# B&R Automation Studio project testovaci_pneu_stan
Automation Studio 4.9

## Configuration Config1

### Acp10map.ncm - 4PPC70_0702_20B/Motion/Acp10map.ncm
```
NcMapping (NcSwId=Acp10)
  NcObject gAxis01 (ModuleId=8V1010.50-2, Type=ncAXIS, Channel=1, AcoposSimulation=Off, InitParameter=gAxis01i, AcoposParameter=gAxis01a, Disabled=FALSE, ModuleDisabled=FALSE)
  NcObject 8V1010.50-2_ncV_AXIS1 (ModuleId=8V1010.50-2, Type=ncV_AXIS, Channel=1, Disabled=TRUE, ModuleDisabled=FALSE)
  NcObject gAxis02 (ModuleId=8V1010.50-2a, Type=ncAXIS, Channel=1, AcoposSimulation=Off, InitParameter=gAxis02i, AcoposParameter=gAxis02a, Disabled=FALSE, ModuleDisabled=FALSE)
  NcObject 8V1010.50-2a_ncV_AXIS1 (ModuleId=8V1010.50-2a, Type=ncV_AXIS, Channel=1, Disabled=TRUE, ModuleDisabled=FALSE)
```

## Logical view

### Library Logical/Libraries/pomoc_lib

#### pomoc_lib.fun
```iecst
FUNCTION_BLOCK cyklovac_b
	VAR_INPUT
		ssMethodType :  SINT;
		krok_tlaku :  REAL :=  0; (*riadok matice zasobujucej cyklovac*)
	END_VAR
	VAR_OUTPUT
		tlak_blue_1 :  REAL :=  0; (*blue_tlak*)
		tlak_green_1 :  REAL :=  0; (**)
		tlak_yellow_1 :  REAL :=  0; (**)
	END_VAR
	VAR
		bur_B_cyklovac_BB_T :  B_cyklovac_BB_T;
		bur_cyklovac_BB :  tag_RTM_cyklovac_BB_T;
	END_VAR
END_FUNCTION_BLOCK
```

#### cyklovac_BB.h
```c
/*
 * cyklovac_BB.h
 *
 * Academic License - for use in teaching, academic research, and meeting
 * course requirements at degree granting institutions only.  Not for
 * government, commercial, or other organizational use.
 *
 * Code generation for model "cyklovac_BB".
 *
 * Model version              : 1.8
 * Simulink Coder version : 9.6 (R2021b) 14-May-2021
 * C source code generated on : Thu Mar 17 07:18:42 2022
 *
 * Target selection: bur_grt.tlc
 * Note: GRT includes extra infrastructure and instrumentation for prototyping
 * Embedded hardware selection: Intel->x86/Pentium
 * Code generation objectives: Unspecified
 * Validation result: Not run
 */

#ifndef RTW_HEADER_cyklovac_BB_h_
#define RTW_HEADER_cyklovac_BB_h_
#include <stddef.h>
#include <string.h>
#ifndef cyklovac_BB_COMMON_INCLUDES_
#define cyklovac_BB_COMMON_INCLUDES_
#include <stdlib.h>
#include "rtwtypes.h"
#include "rtw_continuous.h"
#include "rtw_solver.h"
#endif                                 /* cyklovac_BB_COMMON_INCLUDES_ */

#include "cyklovac_BB_types.h"
#include "pomoc_lib.h"
/* Beginning of Dynamic TypeDefs: */
/* End of Dynamic TypeDefs: */
#ifndef MIN
#define MIN(a,b)	((a) < (b) ? (a) : (b))
#endif

#ifndef MAX
#define MAX(a,b)	((a) > (b) ? (a) : (b))
#endif

#ifndef AST_ROUND
#define AST_ROUND(x) ((x)>=0?(long long)((x)+0.5):(long long)((x)-0.5))
#endif

/* Shared type includes */
#include "multiword_types.h"
#include "rt_defines.h"

/* Macros for accessing real-time model data structure */
#ifndef rtmGetBlockIO
#define rtmGetBlockIO(rtm)             ((rtm)->blockIO)
#endif

#ifndef rtmSetBlockIO
#define rtmSetBlockIO(rtm, val)        ((rtm)->blockIO = (val))
#endif

#ifndef rtmGetErrorStatus
#define rtmGetErrorStatus(rtm)         ((rtm)->errorStatus)
#endif

#ifndef rtmSetErrorStatus
#define rtmSetErrorStatus(rtm, val)    ((rtm)->errorStatus = (val))
#endif

#define cyklovac_BB_M_TYPE             RT_MODEL_cyklovac_BB_T

/* Block signals (default storage) */

/* Constant parameters (default storage) */

/* Real-time Model Data Structure */

/* External data declarations for dependent source files */
extern const char *RT_MEMORY_ALLOCATION_ERROR;

/* Constant parameters (default storage) */
extern const ConstP_cyklovac_BB_T cyklovac_BB_ConstP;

/* Model entry point functions */
extern void cyklovac_BB_initializeMemory(RT_MODEL_cyklovac_BB_T * const cyklovac_BB_M, struct cyklovac_b* inst);
extern void cyklovac_BB_initialize(RT_MODEL_cyklovac_BB_T *const cyklovac_BB_M, struct cyklovac_b* inst);
extern void cyklovac_BB_step(RT_MODEL_cyklovac_BB_T *const cyklovac_BB_M, struct cyklovac_b* inst);
extern void cyklovac_BB_terminate(RT_MODEL_cyklovac_BB_T * cyklovac_BB_M, struct cyklovac_b* inst);

/*-
 * The generated code includes comments that allow you to trace directly
 * back to the appropriate location in the model.  The basic format
 * is <system>/block_name, where system is the system number (uniquely
 * assigned by Simulink) and block_name is the name of the block.
 *
 * Use the MATLAB hilite_system command to trace the generated code back
 * to the model.  For example,
 *
 * hilite_system('<S3>')    - opens system 3
 * hilite_system('<S3>/Kp') - opens and selects block Kp which resides in S3
 *
 * Here is the system hierarchy for this model
 *
 * '<Root>' : 'cyklovac_BB'
 * '<S1>'   : 'cyklovac_BB/MATLAB Function'
 */
#endif                                 /* RTW_HEADER_cyklovac_BB_h_ */
```

#### cyklovac_BB_types.h
```c
/*
 * cyklovac_BB_types.h
 *
 * Academic License - for use in teaching, academic research, and meeting
 * course requirements at degree granting institutions only.  Not for
 * government, commercial, or other organizational use.
 *
 * Code generation for model "cyklovac_BB".
 *
 * Model version              : 1.8
 * Simulink Coder version : 9.6 (R2021b) 14-May-2021
 * C source code generated on : Thu Mar 17 07:18:42 2022
 *
 * Target selection: bur_grt.tlc
 * Note: GRT includes extra infrastructure and instrumentation for prototyping
 * Embedded hardware selection: Intel->x86/Pentium
 * Code generation objectives: Unspecified
 * Validation result: Not run
 */

#ifndef RTW_HEADER_cyklovac_BB_types_h_
#define RTW_HEADER_cyklovac_BB_types_h_

/* Model Code Variants */

/* Forward declaration for rtModel */

#endif                                 /* RTW_HEADER_cyklovac_BB_types_h_ */
```

#### multiword_types.h
```c
/*
 * multiword_types.h
 *
 * Academic License - for use in teaching, academic research, and meeting
 * course requirements at degree granting institutions only.  Not for
 * government, commercial, or other organizational use.
 *
 * Code generation for model "cyklovac_BB".
 *
 * Model version              : 1.8
 * Simulink Coder version : 9.6 (R2021b) 14-May-2021
 * C source code generated on : Thu Mar 17 07:18:42 2022
 *
 * Target selection: bur_grt.tlc
 * Note: GRT includes extra infrastructure and instrumentation for prototyping
 * Embedded hardware selection: Intel->x86/Pentium
 * Code generation objectives: Unspecified
 * Validation result: Not run
 */

#ifndef MULTIWORD_TYPES_H
#define MULTIWORD_TYPES_H
#include "rtwtypes.h"

/*
 * MultiWord supporting definitions
 */
typedef long int long_T;

/*
 * MultiWord types
 */
typedef struct {
  uint32_T chunks[2];
} int64m_T;

typedef struct {
  int64m_T re;
  int64m_T im;
} cint64m_T;

typedef struct {
  uint32_T chunks[2];
} uint64m_T;

typedef struct {
  uint64m_T re;
  uint64m_T im;
} cuint64m_T;

typedef struct {
  uint32_T chunks[3];
} int96m_T;

typedef struct {
  int96m_T re;
  int96m_T im;
} cint96m_T;

typedef struct {
  uint32_T chunks[3];
} uint96m_T;

typedef struct {
  uint96m_T re;
  uint96m_T im;
} cuint96m_T;

typedef struct {
  uint32_T chunks[4];
} int128m_T;

typedef struct {
  int128m_T re;
  int128m_T im;
} cint128m_T;

typedef struct {
  uint32_T chunks[4];
} uint128m_T;

typedef struct {
  uint128m_T re;
  uint128m_T im;
} cuint128m_T;

typedef struct {
  uint32_T chunks[5];
} int160m_T;

typedef struct {
  int160m_T re;
  int160m_T im;
} cint160m_T;

typedef struct {
  uint32_T chunks[5];
} uint160m_T;

typedef struct {
  uint160m_T re;
  uint160m_T im;
} cuint160m_T;

typedef struct {
  uint32_T chunks[6];
} int192m_T;

typedef struct {
  int192m_T re;
  int192m_T im;
} cint192m_T;

typedef struct {
  uint32_T chunks[6];
} uint192m_T;

typedef struct {
  uint192m_T re;
  uint192m_T im;
} cuint192m_T;

typedef struct {
  uint32_T chunks[7];
} int224m_T;

typedef struct {
  int224m_T re;
  int224m_T im;
} cint224m_T;

typedef struct {
  uint32_T chunks[7];
} uint224m_T;

typedef struct {
  uint224m_T re;
  uint224m_T im;
} cuint224m_T;

typedef struct {
  uint32_T chunks[8];
} int256m_T;

typedef struct {
  int256m_T re;
  int256m_T im;
} cint256m_T;

typedef struct {
  uint32_T chunks[8];
} uint256m_T;

typedef struct {
  uint256m_T re;
  uint256m_T im;
} cuint256m_T;

typedef struct {
  uint32_T chunks[9];
} int288m_T;

typedef struct {
  int288m_T re;
  int288m_T im;
} cint288m_T;

typedef struct {
  uint32_T chunks[9];
} uint288m_T;

typedef struct {
  uint288m_T re;
  uint288m_T im;
} cuint288m_T;

typedef struct {
  uint32_T chunks[10];
} int320m_T;

typedef struct {
  int320m_T re;
  int320m_T im;
} cint320m_T;

typedef struct {
  uint32_T chunks[10];
} uint320m_T;

typedef struct {
  uint320m_T re;
  uint320m_T im;
} cuint320m_T;

typedef struct {
  uint32_T chunks[11];
} int352m_T;

typedef struct {
  int352m_T re;
  int352m_T im;
} cint352m_T;

typedef struct {
  uint32_T chunks[11];
} uint352m_T;

typedef struct {
  uint352m_T re;
  uint352m_T im;
} cuint352m_T;

typedef struct {
  uint32_T chunks[12];
} int384m_T;

typedef struct {
  int384m_T re;
  int384m_T im;
} cint384m_T;

typedef struct {
  uint32_T chunks[12];
} uint384m_T;

typedef struct {
  uint384m_T re;
  uint384m_T im;
} cuint384m_T;

typedef struct {
  uint32_T chunks[13];
} int416m_T;

typedef struct {
  int416m_T re;
  int416m_T im;
} cint416m_T;

typedef struct {
  uint32_T chunks[13];
} uint416m_T;

typedef struct {
  uint416m_T re;
  uint416m_T im;
} cuint416m_T;

typedef struct {
  uint32_T chunks[14];
} int448m_T;

typedef struct {
  int448m_T re;
  int448m_T im;
} cint448m_T;

typedef struct {
  uint32_T chunks[14];
} uint448m_T;

typedef struct {
  uint448m_T re;
  uint448m_T im;
} cuint448m_T;

typedef struct {
  uint32_T chunks[15];
} int480m_T;

typedef struct {
  int480m_T re;
  int480m_T im;
} cint480m_T;

typedef struct {
  uint32_T chunks[15];
} uint480m_T;

typedef struct {
  uint480m_T re;
  uint480m_T im;
} cuint480m_T;

typedef struct {
  uint32_T chunks[16];
} int512m_T;

typedef struct {
  int512m_T re;
  int512m_T im;
} cint512m_T;

typedef struct {
  uint32_T chunks[16];
} uint512m_T;

typedef struct {
  uint512m_T re;
  uint512m_T im;
} cuint512m_T;

typedef struct {
  uint32_T chunks[17];
} int544m_T;

typedef struct {
  int544m_T re;
  int544m_T im;
} cint544m_T;

typedef struct {
  uint32_T chunks[17];
} uint544m_T;

typedef struct {
  uint544m_T re;
  uint544m_T im;
} cuint544m_T;

typedef struct {
  uint32_T chunks[18];
} int576m_T;

typedef struct {
  int576m_T re;
  int576m_T im;
} cint576m_T;

typedef struct {
  uint32_T chunks[18];
} uint576m_T;

typedef struct {
  uint576m_T re;
  uint576m_T im;
} cuint576m_T;

typedef struct {
  uint32_T chunks[19];
} int608m_T;

typedef struct {
  int608m_T re;
  int608m_T im;
} cint608m_T;

typedef struct {
  uint32_T chunks[19];
} uint608m_T;

typedef struct {
  uint608m_T re;
  uint608m_T im;
} cuint608m_T;

typedef struct {
  uint32_T chunks[20];
} int640m_T;

typedef struct {
  int640m_T re;
  int640m_T im;
} cint640m_T;

typedef struct {
  uint32_T chunks[20];
} uint640m_T;

typedef struct {
  uint640m_T re;
  uint640m_T im;
} cuint640m_T;

typedef struct {
  uint32_T chunks[21];
} int672m_T;

typedef struct {
  int672m_T re;
  int672m_T im;
} cint672m_T;

typedef struct {
  uint32_T chunks[21];
} uint672m_T;

typedef struct {
  uint672m_T re;
  uint672m_T im;
} cuint672m_T;

typedef struct {
  uint32_T chunks[22];
} int704m_T;

typedef struct {
  int704m_T re;
  int704m_T im;
} cint704m_T;

typedef struct {
  uint32_T chunks[22];
} uint704m_T;

typedef struct {
  uint704m_T re;
  uint704m_T im;
} cuint704m_T;

typedef struct {
  uint32_T chunks[23];
} int736m_T;

typedef struct {
  int736m_T re;
  int736m_T im;
} cint736m_T;

typedef struct {
  uint32_T chunks[23];
} uint736m_T;

typedef struct {
  uint736m_T re;
  uint736m_T im;
} cuint736m_T;

typedef struct {
  uint32_T chunks[24];
} int768m_T;

typedef struct {
  int768m_T re;
  int768m_T im;
} cint768m_T;

typedef struct {
  uint32_T chunks[24];
} uint768m_T;

typedef struct {
  uint768m_T re;
  uint768m_T im;
} cuint768m_T;

typedef struct {
  uint32_T chunks[25];
} int800m_T;

typedef struct {
  int800m_T re;
  int800m_T im;
} cint800m_T;

typedef struct {
  uint32_T chunks[25];
} uint800m_T;

typedef struct {
  uint800m_T re;
  uint800m_T im;
} cuint800m_T;

typedef struct {
  uint32_T chunks[26];
} int832m_T;

typedef struct {
  int832m_T re;
  int832m_T im;
} cint832m_T;

typedef struct {
  uint32_T chunks[26];
} uint832m_T;

typedef struct {
  uint832m_T re;
  uint832m_T im;
} cuint832m_T;

typedef struct {
  uint32_T chunks[27];
} int864m_T;

typedef struct {
  int864m_T re;
  int864m_T im;
} cint864m_T;

typedef struct {
  uint32_T chunks[27];
} uint864m_T;

typedef struct {
  uint864m_T re;
  uint864m_T im;
} cuint864m_T;

typedef struct {
  uint32_T chunks[28];
} int896m_T;

typedef struct {
  int896m_T re;
  int896m_T im;
} cint896m_T;

typedef struct {
  uint32_T chunks[28];
} uint896m_T;

typedef struct {
  uint896m_T re;
  uint896m_T im;
} cuint896m_T;

typedef struct {
  uint32_T chunks[29];
} int928m_T;

typedef struct {
  int928m_T re;
  int928m_T im;
} cint928m_T;

typedef struct {
  uint32_T chunks[29];
} uint928m_T;

typedef struct {
  uint928m_T re;
  uint928m_T im;
} cuint928m_T;

typedef struct {
  uint32_T chunks[30];
} int960m_T;

typedef struct {
  int960m_T re;
  int960m_T im;
} cint960m_T;

typedef struct {
  uint32_T chunks[30];
} uint960m_T;

typedef struct {
  uint960m_T re;
  uint960m_T im;
} cuint960m_T;

typedef struct {
  uint32_T chunks[31];
} int992m_T;

typedef struct {
  int992m_T re;
  int992m_T im;
} cint992m_T;

typedef struct {
  uint32_T chunks[31];
} uint992m_T;

typedef struct {
  uint992m_T re;
  uint992m_T im;
} cuint992m_T;

typedef struct {
  uint32_T chunks[32];
} int1024m_T;

typedef struct {
  int1024m_T re;
  int1024m_T im;
} cint1024m_T;

typedef struct {
  uint32_T chunks[32];
} uint1024m_T;

typedef struct {
  uint1024m_T re;
  uint1024m_T im;
} cuint1024m_T;

typedef struct {
  uint32_T chunks[33];
} int1056m_T;

typedef struct {
  int1056m_T re;
  int1056m_T im;
} cint1056m_T;

typedef struct {
  uint32_T chunks[33];
} uint1056m_T;

typedef struct {
  uint1056m_T re;
  uint1056m_T im;
} cuint1056m_T;

typedef struct {
  uint32_T chunks[34];
} int1088m_T;

typedef struct {
  int1088m_T re;
  int1088m_T im;
} cint1088m_T;

typedef struct {
  uint32_T chunks[34];
} uint1088m_T;

typedef struct {
  uint1088m_T re;
  uint1088m_T im;
} cuint1088m_T;

typedef struct {
  uint32_T chunks[35];
} int1120m_T;

typedef struct {
  int1120m_T re;
  int1120m_T im;
} cint1120m_T;

typedef struct {
  uint32_T chunks[35];
} uint1120m_T;

typedef struct {
  uint1120m_T re;
  uint1120m_T im;
} cuint1120m_T;

typedef struct {
  uint32_T chunks[36];
} int1152m_T;

typedef struct {
  int1152m_T re;
  int1152m_T im;
} cint1152m_T;

typedef struct {
  uint32_T chunks[36];
} uint1152m_T;

typedef struct {
  uint1152m_T re;
  uint1152m_T im;
} cuint1152m_T;

typedef struct {
  uint32_T chunks[37];
} int1184m_T;

typedef struct {
  int1184m_T re;
  int1184m_T im;
} cint1184m_T;

typedef struct {
  uint32_T chunks[37];
} uint1184m_T;

typedef struct {
  uint1184m_T re;
  uint1184m_T im;
} cuint1184m_T;

typedef struct {
  uint32_T chunks[38];
} int1216m_T;

typedef struct {
  int1216m_T re;
  int1216m_T im;
} cint1216m_T;

typedef struct {
  uint32_T chunks[38];
} uint1216m_T;

typedef struct {
  uint1216m_T re;
  uint1216m_T im;
} cuint1216m_T;

typedef struct {
  uint32_T chunks[39];
} int1248m_T;

typedef struct {
  int1248m_T re;
  int1248m_T im;
} cint1248m_T;

typedef struct {
  uint32_T chunks[39];
} uint1248m_T;

typedef struct {
  uint1248m_T re;
  uint1248m_T im;
} cuint1248m_T;

typedef struct {
  uint32_T chunks[40];
} int1280m_T;

typedef struct {
  int1280m_T re;
  int1280m_T im;
} cint1280m_T;

typedef struct {
  uint32_T chunks[40];
} uint1280m_T;

typedef struct {
  uint1280m_T re;
  uint1280m_T im;
} cuint1280m_T;

typedef struct {
  uint32_T chunks[41];
} int1312m_T;

typedef struct {
  int1312m_T re;
  int1312m_T im;
} cint1312m_T;

typedef struct {
  uint32_T chunks[41];
} uint1312m_T;

typedef struct {
  uint1312m_T re;
  uint1312m_T im;
} cuint1312m_T;

typedef struct {
  uint32_T chunks[42];
} int1344m_T;

typedef struct {
  int1344m_T re;
  int1344m_T im;
} cint1344m_T;

typedef struct {
  uint32_T chunks[42];
} uint1344m_T;

typedef struct {
  uint1344m_T re;
  uint1344m_T im;
} cuint1344m_T;

typedef struct {
  uint32_T chunks[43];
} int1376m_T;

typedef struct {
  int1376m_T re;
  int1376m_T im;
} cint1376m_T;

typedef struct {
  uint32_T chunks[43];
} uint1376m_T;

typedef struct {
  uint1376m_T re;
  uint1376m_T im;
} cuint1376m_T;

typedef struct {
  uint32_T chunks[44];
} int1408m_T;

typedef struct {
  int1408m_T re;
  int1408m_T im;
} cint1408m_T;

typedef struct {
  uint32_T chunks[44];
} uint1408m_T;

typedef struct {
  uint1408m_T re;
  uint1408m_T im;
} cuint1408m_T;

typedef struct {
  uint32_T chunks[45];
} int1440m_T;

typedef struct {
  int1440m_T re;
  int1440m_T im;
} cint1440m_T;

typedef struct {
  uint32_T chunks[45];
} uint1440m_T;

typedef struct {
  uint1440m_T re;
  uint1440m_T im;
} cuint1440m_T;

typedef struct {
  uint32_T chunks[46];
} int1472m_T;

typedef struct {
  int1472m_T re;
  int1472m_T im;
} cint1472m_T;

typedef struct {
  uint32_T chunks[46];
} uint1472m_T;

typedef struct {
  uint1472m_T re;
  uint1472m_T im;
} cuint1472m_T;

typedef struct {
  uint32_T chunks[47];
} int1504m_T;

typedef struct {
  int1504m_T re;
  int1504m_T im;
} cint1504m_T;

typedef struct {
  uint32_T chunks[47];
} uint1504m_T;

typedef struct {
  uint1504m_T re;
  uint1504m_T im;
} cuint1504m_T;

typedef struct {
  uint32_T chunks[48];
} int1536m_T;

typedef struct {
  int1536m_T re;
  int1536m_T im;
} cint1536m_T;

typedef struct {
  uint32_T chunks[48];
} uint1536m_T;

typedef struct {
  uint1536m_T re;
  uint1536m_T im;
} cuint1536m_T;

typedef struct {
  uint32_T chunks[49];
} int1568m_T;

typedef struct {
  int1568m_T re;
  int1568m_T im;
} cint1568m_T;

typedef struct {
  uint32_T chunks[49];
} uint1568m_T;

typedef struct {
  uint1568m_T re;
  uint1568m_T im;
} cuint1568m_T;

typedef struct {
  uint32_T chunks[50];
} int1600m_T;

typedef struct {
  int1600m_T re;
  int1600m_T im;
} cint1600m_T;

typedef struct {
  uint32_T chunks[50];
} uint1600m_T;

typedef struct {
  uint1600m_T re;
  uint1600m_T im;
} cuint1600m_T;

typedef struct {
  uint32_T chunks[51];
} int1632m_T;

typedef struct {
  int1632m_T re;
  int1632m_T im;
} cint1632m_T;

typedef struct {
  uint32_T chunks[51];
} uint1632m_T;

typedef struct {
  uint1632m_T re;
  uint1632m_T im;
} cuint1632m_T;

typedef struct {
  uint32_T chunks[52];
} int1664m_T;

typedef struct {
  int1664m_T re;
  int1664m_T im;
} cint1664m_T;

typedef struct {
  uint32_T chunks[52];
} uint1664m_T;

typedef struct {
  uint1664m_T re;
  uint1664m_T im;
} cuint1664m_T;

typedef struct {
  uint32_T chunks[53];
} int1696m_T;

typedef struct {
  int1696m_T re;
  int1696m_T im;
} cint1696m_T;

typedef struct {
  uint32_T chunks[53];
} uint1696m_T;

typedef struct {
  uint1696m_T re;
  uint1696m_T im;
} cuint1696m_T;

typedef struct {
  uint32_T chunks[54];
} int1728m_T;

typedef struct {
  int1728m_T re;
  int1728m_T im;
} cint1728m_T;

typedef struct {
  uint32_T chunks[54];
} uint1728m_T;

typedef struct {
  uint1728m_T re;
  uint1728m_T im;
} cuint1728m_T;

typedef struct {
  uint32_T chunks[55];
} int1760m_T;

typedef struct {
  int1760m_T re;
  int1760m_T im;
} cint1760m_T;

typedef struct {
  uint32_T chunks[55];
} uint1760m_T;

typedef struct {
  uint1760m_T re;
  uint1760m_T im;
} cuint1760m_T;

typedef struct {
  uint32_T chunks[56];
} int1792m_T;

typedef struct {
  int1792m_T re;
  int1792m_T im;
} cint1792m_T;

typedef struct {
  uint32_T chunks[56];
} uint1792m_T;

typedef struct {
  uint1792m_T re;
  uint1792m_T im;
} cuint1792m_T;

typedef struct {
  uint32_T chunks[57];
} int1824m_T;

typedef struct {
  int1824m_T re;
  int1824m_T im;
} cint1824m_T;

typedef struct {
  uint32_T chunks[57];
} uint1824m_T;

typedef struct {
  uint1824m_T re;
  uint1824m_T im;
} cuint1824m_T;

typedef struct {
  uint32_T chunks[58];
} int1856m_T;

typedef struct {
  int1856m_T re;
  int1856m_T im;
} cint1856m_T;

typedef struct {
  uint32_T chunks[58];
} uint1856m_T;

typedef struct {
  uint1856m_T re;
  uint1856m_T im;
} cuint1856m_T;

typedef struct {
  uint32_T chunks[59];
} int1888m_T;

typedef struct {
  int1888m_T re;
  int1888m_T im;
} cint1888m_T;

typedef struct {
  uint32_T chunks[59];
} uint1888m_T;

typedef struct {
  uint1888m_T re;
  uint1888m_T im;
} cuint1888m_T;

typedef struct {
  uint32_T chunks[60];
} int1920m_T;

typedef struct {
  int1920m_T re;
  int1920m_T im;
} cint1920m_T;

typedef struct {
  uint32_T chunks[60];
} uint1920m_T;

typedef struct {
  uint1920m_T re;
  uint1920m_T im;
} cuint1920m_T;

typedef struct {
  uint32_T chunks[61];
} int1952m_T;

typedef struct {
  int1952m_T re;
  int1952m_T im;
} cint1952m_T;

typedef struct {
  uint32_T chunks[61];
} uint1952m_T;

typedef struct {
  uint1952m_T re;
  uint1952m_T im;
} cuint1952m_T;

typedef struct {
  uint32_T chunks[62];
} int1984m_T;

typedef struct {
  int1984m_T re;
  int1984m_T im;
} cint1984m_T;

typedef struct {
  uint32_T chunks[62];
} uint1984m_T;

typedef struct {
  uint1984m_T re;
  uint1984m_T im;
} cuint1984m_T;

typedef struct {
  uint32_T chunks[63];
} int2016m_T;

typedef struct {
  int2016m_T re;
  int2016m_T im;
} cint2016m_T;

typedef struct {
  uint32_T chunks[63];
} uint2016m_T;

typedef struct {
  uint2016m_T re;
  uint2016m_T im;
} cuint2016m_T;

typedef struct {
  uint32_T chunks[64];
} int2048m_T;

typedef struct {
  int2048m_T re;
  int2048m_T im;
} cint2048m_T;

typedef struct {
  uint32_T chunks[64];
} uint2048m_T;

typedef struct {
  uint2048m_T re;
  uint2048m_T im;
} cuint2048m_T;

#endif                                 /* MULTIWORD_TYPES_H */
```

#### cyklovac_BB.c
```c
/*
 * cyklovac_BB.c
 *
 * Academic License - for use in teaching, academic research, and meeting
 * course requirements at degree granting institutions only.  Not for
 * government, commercial, or other organizational use.
 *
 * Code generation for model "cyklovac_BB".
 *
 * Model version              : 1.8
 * Simulink Coder version : 9.6 (R2021b) 14-May-2021
 * C source code generated on : Thu Mar 17 07:18:42 2022
 *
 * Target selection: bur_grt.tlc
 * Note: GRT includes extra infrastructure and instrumentation for prototyping
 * Embedded hardware selection: Intel->x86/Pentium
 * Code generation objectives: Unspecified
 * Validation result: Not run
 */

#include "cyklovac_BB.h"
#include "cyklovac_BB_private.h"

/* Model step function */
void cyklovac_BB_step(RT_MODEL_cyklovac_BB_T *const cyklovac_BB_M, struct cyklovac_b* inst)
{
  B_cyklovac_BB_T *cyklovac_BB_B = cyklovac_BB_M->blockIO;

  /* S-Function (bur_in): '<Root>/Input' */
  cyklovac_BB_B->Input = inst->krok_tlaku;

  /* Gain: '<Root>/Gain' incorporates:
   *  Constant: '<Root>/Constant'
   *  MATLAB Function: '<Root>/MATLAB Function'
   */
  cyklovac_BB_B->Gain = (real32_T)cyklovac_BB_ConstP.Constant_Value[(int32_T)
    cyklovac_BB_B->Input - 1];

  /* S-Function (bur_out): '<Root>/Output' */
  inst->tlak_blue_1 = cyklovac_BB_B->Gain;

  /* Gain: '<Root>/Gain1' incorporates:
   *  Constant: '<Root>/Constant'
   *  MATLAB Function: '<Root>/MATLAB Function'
   */
  cyklovac_BB_B->Gain1 = (real32_T)cyklovac_BB_ConstP.Constant_Value[(int32_T)
    cyklovac_BB_B->Input + 783];

  /* S-Function (bur_out): '<Root>/Output1' */
  inst->tlak_green_1 = cyklovac_BB_B->Gain1;

  /* Gain: '<Root>/Gain2' incorporates:
   *  Constant: '<Root>/Constant'
   *  MATLAB Function: '<Root>/MATLAB Function'
   */
  cyklovac_BB_B->Gain2 = (real32_T)cyklovac_BB_ConstP.Constant_Value[(int32_T)
    cyklovac_BB_B->Input + 1567];

  /* S-Function (bur_out): '<Root>/Output2' */
  inst->tlak_yellow_1 = cyklovac_BB_B->Gain2;
}

/* Model initialize function */
void cyklovac_BB_initialize(RT_MODEL_cyklovac_BB_T *const cyklovac_BB_M, struct cyklovac_b* inst)
{
  UNUSED_PARAMETER(cyklovac_BB_M);
}

/* Model terminate function */
void cyklovac_BB_terminate(RT_MODEL_cyklovac_BB_T * cyklovac_BB_M, struct cyklovac_b* inst)
{}

/* Model data allocation function */
void cyklovac_BB_initializeMemory(RT_MODEL_cyklovac_BB_T* const cyklovac_BB_M, struct cyklovac_b * inst)
{
  /* block I/O */
  {
  }

  {
    B_cyklovac_BB_T *cyklovac_BB_B = cyklovac_BB_M->blockIO;

    /* block I/O */
    {
      cyklovac_BB_B->Input = 0.0F;
      cyklovac_BB_B->Gain = 0.0F;
      cyklovac_BB_B->Gain1 = 0.0F;
      cyklovac_BB_B->Gain2 = 0.0F;
    }
  }

}
```

#### cyklovac_BB_data.c
```c
/*
 * cyklovac_BB_data.c
 *
 * Academic License - for use in teaching, academic research, and meeting
 * course requirements at degree granting institutions only.  Not for
 * government, commercial, or other organizational use.
 *
 * Code generation for model "cyklovac_BB".
 *
 * Model version              : 1.8
 * Simulink Coder version : 9.6 (R2021b) 14-May-2021
 * C source code generated on : Thu Mar 17 07:18:42 2022
 *
 * Target selection: bur_grt.tlc
 * Note: GRT includes extra infrastructure and instrumentation for prototyping
 * Embedded hardware selection: Intel->x86/Pentium
 * Code generation objectives: Unspecified
 * Validation result: Not run
 */

#include "cyklovac_BB.h"
#include "cyklovac_BB_private.h"

/* Constant parameters (default storage) */
const ConstP_cyklovac_BB_T cyklovac_BB_ConstP = {
  /* Expression: tlaky_upravene
   * Referenced by: '<Root>/Constant'
   */
  { 0.25, 0.25, 0.25, 0.25, 0.25, 0.25, 0.25, 0.25, 0.25, 0.25, 0.25, 0.25, 0.25,
    0.25, 0.25, 0.25, 0.25, 0.25, 0.25, 0.25, 0.25, 0.25, 0.25, 0.25, 0.25, 0.25,
    0.25, 0.25, 0.25, 0.25, 0.25, 0.25, 0.25, 0.25, 0.25, 0.25, 0.25, 0.25, 0.25,
    0.25, 0.25, 0.25, 0.25, 0.25, 0.25, 0.25, 0.25, 0.25, 0.25, 0.25, 0.25, 0.25,
    0.25, 0.25, 0.25, 0.25, 0.25, 0.25, 0.25, 0.25, 0.25, 0.25, 0.25, 0.25, 0.25,
    0.25, 0.25, 0.25, 0.25, 0.25, 0.25, 0.25, 0.25, 0.25, 0.25, 0.25, 0.25, 0.25,
    0.25, 0.25, 0.25, 0.25, 0.25, 0.25, 0.25, 0.25, 0.25, 0.25, 0.25, 0.25, 0.25,
    0.25, 0.25, 0.25, 0.25, 0.25, 0.25, 0.25, 0.25, 0.25, 0.75, 0.75, 0.75, 0.75,
    0.75, 0.75, 0.75, 0.75, 0.75, 0.75, 0.75, 0.75, 0.75, 0.75, 0.75, 0.75, 0.75,
    0.75, 0.75, 0.75, 0.75, 0.75, 0.75, 0.75, 0.75, 0.75, 0.75, 0.75, 0.75, 0.75,
    0.75, 0.75, 0.75, 0.75, 0.75, 0.75, 0.75, 0.75, 0.75, 0.75, 0.75, 0.75, 0.75,
    0.75, 0.75, 0.75, 0.75, 0.75, 0.75, 0.75, 0.75, 0.75, 0.75, 0.75, 0.75, 0.75,
    0.75, 0.75, 0.75, 0.75, 0.75, 0.75, 0.75, 0.75, 0.75, 0.75, 0.75, 0.75, 0.75,
    0.75, 0.75, 0.75, 0.75, 0.75, 0.75, 0.75, 0.75, 0.75, 0.75, 0.75, 0.75, 0.75,
    0.75, 0.75, 0.75, 0.75, 0.75, 0.75, 0.75, 0.75, 0.75, 0.75, 0.75, 0.75, 0.75,
    0.75, 0.75, 0.75, 0.75, 0.75, 1.25, 1.25, 1.25, 1.25, 1.25, 1.25, 1.25, 1.25,
    1.25, 1.25, 1.25, 1.25, 1.25, 1.25, 1.25, 1.25, 1.25, 1.25, 1.25, 1.25, 1.25,
    1.25, 1.25, 1.25, 1.25, 1.25, 1.25, 1.25, 1.25, 1.25, 1.25, 1.25, 1.25, 1.25,
    1.25, 1.25, 1.25, 1.25, 1.25, 1.25, 1.25, 1.25, 1.25, 1.25, 1.25, 1.25, 1.25,
    1.25, 1.25, 1.25, 1.25, 1.25, 1.25, 1.25, 1.25, 1.25, 1.25, 1.25, 1.25, 1.25,
    1.25, 1.25, 1.25, 1.25, 1.25, 1.25, 1.25, 1.25, 1.25, 1.25, 1.25, 1.25, 1.25,
    1.25, 1.25, 1.25, 1.25, 1.25, 1.25, 1.25, 1.25, 1.25, 1.25, 1.25, 1.25, 1.25,
    1.25, 1.25, 1.25, 1.25, 1.25, 1.25, 1.25, 1.25, 1.25, 1.25, 1.25, 1.25, 1.25,
    1.25, 1.75, 1.75, 1.75, 1.75, 1.75, 1.75, 1.75, 1.75, 1.75, 1.75, 1.75, 1.75,
    1.75, 1.75, 1.75, 1.75, 1.75, 1.75, 1.75, 1.75, 1.75, 1.75, 1.75, 1.75, 1.75,
    1.75, 1.75, 1.75, 1.75, 1.75, 1.75, 1.75, 1.75, 1.75, 1.75, 1.75, 1.75, 1.75,
    1.75, 1.75, 1.75, 1.75, 1.75, 1.75, 1.75, 1.75, 1.75, 1.75, 1.75, 1.75, 1.75,
    1.75, 1.75, 1.75, 1.75, 1.75, 1.75, 1.75, 1.75, 1.75, 1.75, 1.75, 1.75, 1.75,
    1.75, 1.75, 1.75, 1.75, 1.75, 1.75, 1.75, 1.75, 1.75, 1.75, 1.75, 1.75, 1.75,
    1.75, 1.75, 1.75, 1.75, 1.75, 1.75, 1.75, 1.75, 1.75, 1.75, 1.75, 1.75, 1.75,
    1.75, 1.75, 1.75, 1.75, 1.75, 1.75, 1.75, 1.75, 1.75, 1.75, 2.25, 2.25, 2.25,
    2.25, 2.25, 2.25, 2.25, 2.25, 2.25, 2.25, 2.25, 2.25, 2.25, 2.25, 2.25, 2.25,
    2.25, 2.25, 2.25, 2.25, 2.25, 2.25, 2.25, 2.25, 2.25, 2.25, 2.25, 2.25, 2.25,
    2.25, 2.25, 2.25, 2.25, 2.25, 2.25, 2.25, 2.25, 2.25, 2.25, 2.25, 2.25, 2.25,
    2.25, 2.25, 2.25, 2.25, 2.25, 2.25, 2.25, 2.25, 2.25, 2.25, 2.25, 2.25, 2.25,
    2.25, 2.25, 2.25, 2.25, 2.25, 2.25, 2.25, 2.25, 2.25, 2.75, 2.75, 2.75, 2.75,
    2.75, 2.75, 2.75, 2.75, 2.75, 2.75, 2.75, 2.75, 2.75, 2.75, 2.75, 2.75, 2.75,
    2.75, 2.75, 2.75, 2.75, 2.75, 2.75, 2.75, 2.75, 2.75, 2.75, 2.75, 2.75, 2.75,
    2.75, 2.75, 2.75, 2.75, 2.75, 2.75, 2.75, 2.75, 2.75, 2.75, 2.75, 2.75, 2.75,
    2.75, 2.75, 2.75, 2.75, 2.75, 2.75, 2.75, 2.75, 2.75, 2.75, 2.75, 2.75, 2.75,
    2.75, 2.75, 2.75, 2.75, 2.75, 2.75, 2.75, 2.75, 3.25, 3.25, 3.25, 3.25, 3.25,
    3.25, 3.25, 3.25, 3.25, 3.25, 3.25, 3.25, 3.25, 3.25, 3.25, 3.25, 3.25, 3.25,
    3.25, 3.25, 3.25, 3.25, 3.25, 3.25, 3.25, 3.25, 3.25, 3.25, 3.25, 3.25, 3.25,
    3.25, 3.25, 3.25, 3.25, 3.25, 3.25, 3.25, 3.25, 3.25, 3.25, 3.25, 3.25, 3.25,
    3.25, 3.25, 3.25, 3.25, 3.25, 3.25, 3.25, 3.25, 3.25, 3.25, 3.25, 3.25, 3.25,
    3.25, 3.25, 3.25, 3.25, 3.25, 3.25, 3.25, 3.75, 3.75, 3.75, 3.75, 3.75, 3.75,
    3.75, 3.75, 3.75, 3.75, 3.75, 3.75, 3.75, 3.75, 3.75, 3.75, 3.75, 3.75, 3.75,
    3.75, 3.75, 3.75, 3.75, 3.75, 3.75, 3.75, 3.75, 3.75, 3.75, 3.75, 3.75, 3.75,
    3.75, 3.75, 3.75, 3.75, 3.75, 3.75, 3.75, 3.75, 3.75, 3.75, 3.75, 3.75, 3.75,
    3.75, 3.75, 3.75, 3.75, 3.75, 3.75, 3.75, 3.75, 3.75, 3.75, 3.75, 3.75, 3.75,
    3.75, 3.75, 3.75, 3.75, 3.75, 3.75, 4.25, 4.25, 4.25, 4.25, 4.25, 4.25, 4.25,
    4.25, 4.25, 4.25, 4.25, 4.25, 4.25, 4.25, 4.25, 4.25, 4.25, 4.25, 4.25, 4.25,
    4.25, 4.25, 4.25, 4.25, 4.25, 4.25, 4.25, 4.25, 4.25, 4.25, 4.25, 4.25, 4.25,
    4.25, 4.25, 4.25, 4.25, 4.25, 4.25, 4.25, 4.25, 4.25, 4.25, 4.25, 4.25, 4.25,
    4.25, 4.25, 4.25, 4.25, 4.25, 4.25, 4.25, 4.25, 4.25, 4.25, 4.25, 4.25, 4.25,
    4.25, 4.25, 4.25, 4.25, 4.25, 4.75, 4.75, 4.75, 4.75, 4.75, 4.75, 4.75, 4.75,
    4.75, 4.75, 4.75, 4.75, 4.75, 4.75, 4.75, 4.75, 4.75, 4.75, 4.75, 4.75, 4.75,
    4.75, 4.75, 4.75, 4.75, 4.75, 4.75, 4.75, 4.75, 4.75, 4.75, 4.75, 4.75, 4.75,
    4.75, 4.75, 4.75, 4.75, 4.75, 4.75, 4.75, 4.75, 4.75, 4.75, 4.75, 4.75, 4.75,
    4.75, 4.75, 4.75, 4.75, 4.75, 4.75, 4.75, 4.75, 4.75, 4.75, 4.75, 4.75, 4.75,
    4.75, 4.75, 4.75, 4.75, 0.25, 0.25, 0.25, 0.25, 0.25, 0.25, 0.25, 0.25, 0.25,
    0.25, 0.75, 0.75, 0.75, 0.75, 0.75, 0.75, 0.75, 0.75, 0.75, 0.75, 1.25, 1.25,
    1.25, 1.25, 1.25, 1.25, 1.25, 1.25, 1.25, 1.25, 1.75, 1.75, 1.75, 1.75, 1.75,
    1.75, 1.75, 1.75, 1.75, 1.75, 2.25, 2.25, 2.25, 2.25, 2.25, 2.25, 2.25, 2.25,
    2.25, 2.25, 2.75, 2.75, 2.75, 2.75, 2.75, 2.75, 2.75, 2.75, 2.75, 2.75, 3.25,
    3.25, 3.25, 3.25, 3.25, 3.25, 3.25, 3.25, 3.25, 3.25, 3.75, 3.75, 3.75, 3.75,
    3.75, 3.75, 3.75, 3.75, 3.75, 3.75, 4.25, 4.25, 4.25, 4.25, 4.25, 4.25, 4.25,
    4.25, 4.25, 4.25, 4.75, 4.75, 4.75, 4.75, 4.75, 4.75, 4.75, 4.75, 4.75, 4.75,
    0.25, 0.25, 0.25, 0.25, 0.25, 0.25, 0.25, 0.25, 0.25, 0.25, 0.75, 0.75, 0.75,
    0.75, 0.75, 0.75, 0.75, 0.75, 0.75, 0.75, 1.25, 1.25, 1.25, 1.25, 1.25, 1.25,
    1.25, 1.25, 1.25, 1.25, 1.75, 1.75, 1.75, 1.75, 1.75, 1.75, 1.75, 1.75, 1.75,
    1.75, 2.25, 2.25, 2.25, 2.25, 2.25, 2.25, 2.25, 2.25, 2.25, 2.25, 2.75, 2.75,
    2.75, 2.75, 2.75, 2.75, 2.75, 2.75, 2.75, 2.75, 3.25, 3.25, 3.25, 3.25, 3.25,
    3.25, 3.25, 3.25, 3.25, 3.25, 3.75, 3.75, 3.75, 3.75, 3.75, 3.75, 3.75, 3.75,
    3.75, 3.75, 4.25, 4.25, 4.25, 4.25, 4.25, 4.25, 4.25, 4.25, 4.25, 4.25, 4.75,
    4.75, 4.75, 4.75, 4.75, 4.75, 4.75, 4.75, 4.75, 4.75, 0.25, 0.25, 0.25, 0.25,
    0.25, 0.25, 0.25, 0.25, 0.25, 0.25, 0.75, 0.75, 0.75, 0.75, 0.75, 0.75, 0.75,
    0.75, 0.75, 0.75, 1.25, 1.25, 1.25, 1.25, 1.25, 1.25, 1.25, 1.25, 1.25, 1.25,
    1.75, 1.75, 1.75, 1.75, 1.75, 1.75, 1.75, 1.75, 1.75, 1.75, 2.25, 2.25, 2.25,
    2.25, 2.25, 2.25, 2.25, 2.25, 2.25, 2.25, 2.75, 2.75, 2.75, 2.75, 2.75, 2.75,
    2.75, 2.75, 2.75, 2.75, 3.25, 3.25, 3.25, 3.25, 3.25, 3.25, 3.25, 3.25, 3.25,
    3.25, 3.75, 3.75, 3.75, 3.75, 3.75, 3.75, 3.75, 3.75, 3.75, 3.75, 4.25, 4.25,
    4.25, 4.25, 4.25, 4.25, 4.25, 4.25, 4.25, 4.25, 4.75, 4.75, 4.75, 4.75, 4.75,
    4.75, 4.75, 4.75, 4.75, 4.75, 0.25, 0.25, 0.25, 0.25, 0.25, 0.25, 0.25, 0.25,
    0.25, 0.25, 0.75, 0.75, 0.75, 0.75, 0.75, 0.75, 0.75, 0.75, 0.75, 0.75, 1.25,
    1.25, 1.25, 1.25, 1.25, 1.25, 1.25, 1.25, 1.25, 1.25, 1.75, 1.75, 1.75, 1.75,
    1.75, 1.75, 1.75, 1.75, 1.75, 1.75, 2.25, 2.25, 2.25, 2.25, 2.25, 2.25, 2.25,
    2.25, 2.25, 2.25, 2.75, 2.75, 2.75, 2.75, 2.75, 2.75, 2.75, 2.75, 2.75, 2.75,
    3.25, 3.25, 3.25, 3.25, 3.25, 3.25, 3.25, 3.25, 3.25, 3.25, 3.75, 3.75, 3.75,
    3.75, 3.75, 3.75, 3.75, 3.75, 3.75, 3.75, 4.25, 4.25, 4.25, 4.25, 4.25, 4.25,
    4.25, 4.25, 4.25, 4.25, 4.75, 4.75, 4.75, 4.75, 4.75, 4.75, 4.75, 4.75, 4.75,
    4.75, 0.25, 0.25, 0.25, 0.25, 0.25, 0.25, 0.25, 0.25, 0.25, 0.25, 0.75, 0.75,
    0.75, 0.75, 0.75, 0.75, 0.75, 0.75, 0.75, 0.75, 1.25, 1.25, 1.25, 1.25, 1.25,
    1.25, 1.25, 1.25, 1.25, 1.25, 1.75, 1.75, 1.75, 1.75, 1.75, 1.75, 1.75, 1.75,
    1.75, 1.75, 2.25, 2.25, 2.25, 2.25, 2.75, 2.75, 2.75, 2.75, 3.25, 3.25, 3.25,
    3.25, 3.75, 3.75, 3.75, 3.75, 4.25, 4.25, 4.25, 4.25, 4.75, 4.75, 4.75, 4.75,
    0.25, 0.25, 0.25, 0.25, 0.25, 0.25, 0.25, 0.25, 0.25, 0.25, 0.75, 0.75, 0.75,
    0.75, 0.75, 0.75, 0.75, 0.75, 0.75, 0.75, 1.25, 1.25, 1.25, 1.25, 1.25, 1.25,
    1.25, 1.25, 1.25, 1.25, 1.75, 1.75, 1.75, 1.75, 1.75, 1.75, 1.75, 1.75, 1.75,
    1.75, 2.25, 2.25, 2.25, 2.25, 2.75, 2.75, 2.75, 2.75, 3.25, 3.25, 3.25, 3.25,
    3.75, 3.75, 3.75, 3.75, 4.25, 4.25, 4.25, 4.25, 4.75, 4.75, 4.75, 4.75, 0.25,
    0.25, 0.25, 0.25, 0.25, 0.25, 0.25, 0.25, 0.25, 0.25, 0.75, 0.75, 0.75, 0.75,
    0.75, 0.75, 0.75, 0.75, 0.75, 0.75, 1.25, 1.25, 1.25, 1.25, 1.25, 1.25, 1.25,
    1.25, 1.25, 1.25, 1.75, 1.75, 1.75, 1.75, 1.75, 1.75, 1.75, 1.75, 1.75, 1.75,
    2.25, 2.25, 2.25, 2.25, 2.75, 2.75, 2.75, 2.75, 3.25, 3.25, 3.25, 3.25, 3.75,
    3.75, 3.75, 3.75, 4.25, 4.25, 4.25, 4.25, 4.75, 4.75, 4.75, 4.75, 0.25, 0.25,
    0.25, 0.25, 0.25, 0.25, 0.25, 0.25, 0.25, 0.25, 0.75, 0.75, 0.75, 0.75, 0.75,
    0.75, 0.75, 0.75, 0.75, 0.75, 1.25, 1.25, 1.25, 1.25, 1.25, 1.25, 1.25, 1.25,
    1.25, 1.25, 1.75, 1.75, 1.75, 1.75, 1.75, 1.75, 1.75, 1.75, 1.75, 1.75, 2.25,
    2.25, 2.25, 2.25, 2.75, 2.75, 2.75, 2.75, 3.25, 3.25, 3.25, 3.25, 3.75, 3.75,
    3.75, 3.75, 4.25, 4.25, 4.25, 4.25, 4.75, 4.75, 4.75, 4.75, 0.25, 0.25, 0.25,
    0.25, 0.25, 0.25, 0.25, 0.25, 0.25, 0.25, 0.75, 0.75, 0.75, 0.75, 0.75, 0.75,
    0.75, 0.75, 0.75, 0.75, 1.25, 1.25, 1.25, 1.25, 1.25, 1.25, 1.25, 1.25, 1.25,
    1.25, 1.75, 1.75, 1.75, 1.75, 1.75, 1.75, 1.75, 1.75, 1.75, 1.75, 2.25, 2.25,
    2.25, 2.25, 2.75, 2.75, 2.75, 2.75, 3.25, 3.25, 3.25, 3.25, 3.75, 3.75, 3.75,
    3.75, 4.25, 4.25, 4.25, 4.25, 4.75, 4.75, 4.75, 4.75, 0.25, 0.25, 0.25, 0.25,
    0.25, 0.25, 0.25, 0.25, 0.25, 0.25, 0.75, 0.75, 0.75, 0.75, 0.75, 0.75, 0.75,
    0.75, 0.75, 0.75, 1.25, 1.25, 1.25, 1.25, 1.25, 1.25, 1.25, 1.25, 1.25, 1.25,
    1.75, 1.75, 1.75, 1.75, 1.75, 1.75, 1.75, 1.75, 1.75, 1.75, 2.25, 2.25, 2.25,
    2.25, 2.75, 2.75, 2.75, 2.75, 3.25, 3.25, 3.25, 3.25, 3.75, 3.75, 3.75, 3.75,
    4.25, 4.25, 4.25, 4.25, 4.75, 4.75, 4.75, 4.75, 0.25, 0.75, 1.25, 1.75, 2.25,
    2.75, 3.25, 3.75, 4.25, 4.75, 0.25, 0.75, 1.25, 1.75, 2.25, 2.75, 3.25, 3.75,
    4.25, 4.75, 0.25, 0.75, 1.25, 1.75, 2.25, 2.75, 3.25, 3.75, 4.25, 4.75, 0.25,
    0.75, 1.25, 1.75, 2.25, 2.75, 3.25, 3.75, 4.25, 4.75, 0.25, 0.75, 1.25, 1.75,
    2.25, 2.75, 3.25, 3.75, 4.25, 4.75, 0.25, 0.75, 1.25, 1.75, 2.25, 2.75, 3.25,
    3.75, 4.25, 4.75, 0.25, 0.75, 1.25, 1.75, 2.25, 2.75, 3.25, 3.75, 4.25, 4.75,
    0.25, 0.75, 1.25, 1.75, 2.25, 2.75, 3.25, 3.75, 4.25, 4.75, 0.25, 0.75, 1.25,
    1.75, 2.25, 2.75, 3.25, 3.75, 4.25, 4.75, 0.25, 0.75, 1.25, 1.75, 2.25, 2.75,
    3.25, 3.75, 4.25, 4.75, 0.25, 0.75, 1.25, 1.75, 2.25, 2.75, 3.25, 3.75, 4.25,
    4.75, 0.25, 0.75, 1.25, 1.75, 2.25, 2.75, 3.25, 3.75, 4.25, 4.75, 0.25, 0.75,
    1.25, 1.75, 2.25, 2.75, 3.25, 3.75, 4.25, 4.75, 0.25, 0.75, 1.25, 1.75, 2.25,
    2.75, 3.25, 3.75, 4.25, 4.75, 0.25, 0.75, 1.25, 1.75, 2.25, 2.75, 3.25, 3.75,
    4.25, 4.75, 0.25, 0.75, 1.25, 1.75, 2.25, 2.75, 3.25, 3.75, 4.25, 4.75, 0.25,
    0.75, 1.25, 1.75, 2.25, 2.75, 3.25, 3.75, 4.25, 4.75, 0.25, 0.75, 1.25, 1.75,
    2.25, 2.75, 3.25, 3.75, 4.25, 4.75, 0.25, 0.75, 1.25, 1.75, 2.25, 2.75, 3.25,
    3.75, 4.25, 4.75, 0.25, 0.75, 1.25, 1.75, 2.25, 2.75, 3.25, 3.75, 4.25, 4.75,
    0.25, 0.75, 1.25, 1.75, 2.25, 2.75, 3.25, 3.75, 4.25, 4.75, 0.25, 0.75, 1.25,
    1.75, 2.25, 2.75, 3.25, 3.75, 4.25, 4.75, 0.25, 0.75, 1.25, 1.75, 2.25, 2.75,
    3.25, 3.75, 4.25, 4.75, 0.25, 0.75, 1.25, 1.75, 2.25, 2.75, 3.25, 3.75, 4.25,
    4.75, 0.25, 0.75, 1.25, 1.75, 2.25, 2.75, 3.25, 3.75, 4.25, 4.75, 0.25, 0.75,
    1.25, 1.75, 2.25, 2.75, 3.25, 3.75, 4.25, 4.75, 0.25, 0.75, 1.25, 1.75, 2.25,
    2.75, 3.25, 3.75, 4.25, 4.75, 0.25, 0.75, 1.25, 1.75, 2.25, 2.75, 3.25, 3.75,
    4.25, 4.75, 0.25, 0.75, 1.25, 1.75, 2.25, 2.75, 3.25, 3.75, 4.25, 4.75, 0.25,
    0.75, 1.25, 1.75, 2.25, 2.75, 3.25, 3.75, 4.25, 4.75, 0.25, 0.75, 1.25, 1.75,
    2.25, 2.75, 3.25, 3.75, 4.25, 4.75, 0.25, 0.75, 1.25, 1.75, 2.25, 2.75, 3.25,
    3.75, 4.25, 4.75, 0.25, 0.75, 1.25, 1.75, 2.25, 2.75, 3.25, 3.75, 4.25, 4.75,
    0.25, 0.75, 1.25, 1.75, 2.25, 2.75, 3.25, 3.75, 4.25, 4.75, 0.25, 0.75, 1.25,
    1.75, 2.25, 2.75, 3.25, 3.75, 4.25, 4.75, 0.25, 0.75, 1.25, 1.75, 2.25, 2.75,
    3.25, 3.75, 4.25, 4.75, 0.25, 0.75, 1.25, 1.75, 2.25, 2.75, 3.25, 3.75, 4.25,
    4.75, 0.25, 0.75, 1.25, 1.75, 2.25, 2.75, 3.25, 3.75, 4.25, 4.75, 0.25, 0.75,
    1.25, 1.75, 2.25, 2.75, 3.25, 3.75, 4.25, 4.75, 0.25, 0.75, 1.25, 1.75, 2.25,
    2.75, 3.25, 3.75, 4.25, 4.75, 0.25, 0.75, 1.25, 1.75, 2.25, 2.75, 3.25, 3.75,
    4.25, 4.75, 0.25, 0.75, 1.25, 1.75, 2.25, 2.75, 3.25, 3.75, 4.25, 4.75, 0.25,
    0.75, 1.25, 1.75, 2.25, 2.75, 3.25, 3.75, 4.25, 4.75, 0.25, 0.75, 1.25, 1.75,
    2.25, 2.75, 3.25, 3.75, 4.25, 4.75, 0.25, 0.75, 1.25, 1.75, 0.25, 0.75, 1.25,
    1.75, 0.25, 0.75, 1.25, 1.75, 0.25, 0.75, 1.25, 1.75, 0.25, 0.75, 1.25, 1.75,
    0.25, 0.75, 1.25, 1.75, 0.25, 0.75, 1.25, 1.75, 2.25, 2.75, 3.25, 3.75, 4.25,
    4.75, 0.25, 0.75, 1.25, 1.75, 2.25, 2.75, 3.25, 3.75, 4.25, 4.75, 0.25, 0.75,
    1.25, 1.75, 2.25, 2.75, 3.25, 3.75, 4.25, 4.75, 0.25, 0.75, 1.25, 1.75, 2.25,
    2.75, 3.25, 3.75, 4.25, 4.75, 0.25, 0.75, 1.25, 1.75, 0.25, 0.75, 1.25, 1.75,
    0.25, 0.75, 1.25, 1.75, 0.25, 0.75, 1.25, 1.75, 0.25, 0.75, 1.25, 1.75, 0.25,
    0.75, 1.25, 1.75, 0.25, 0.75, 1.25, 1.75, 2.25, 2.75, 3.25, 3.75, 4.25, 4.75,
    0.25, 0.75, 1.25, 1.75, 2.25, 2.75, 3.25, 3.75, 4.25, 4.75, 0.25, 0.75, 1.25,
    1.75, 2.25, 2.75, 3.25, 3.75, 4.25, 4.75, 0.25, 0.75, 1.25, 1.75, 2.25, 2.75,
    3.25, 3.75, 4.25, 4.75, 0.25, 0.75, 1.25, 1.75, 0.25, 0.75, 1.25, 1.75, 0.25,
    0.75, 1.25, 1.75, 0.25, 0.75, 1.25, 1.75, 0.25, 0.75, 1.25, 1.75, 0.25, 0.75,
    1.25, 1.75, 0.25, 0.75, 1.25, 1.75, 2.25, 2.75, 3.25, 3.75, 4.25, 4.75, 0.25,
    0.75, 1.25, 1.75, 2.25, 2.75, 3.25, 3.75, 4.25, 4.75, 0.25, 0.75, 1.25, 1.75,
    2.25, 2.75, 3.25, 3.75, 4.25, 4.75, 0.25, 0.75, 1.25, 1.75, 2.25, 2.75, 3.25,
    3.75, 4.25, 4.75, 0.25, 0.75, 1.25, 1.75, 0.25, 0.75, 1.25, 1.75, 0.25, 0.75,
    1.25, 1.75, 0.25, 0.75, 1.25, 1.75, 0.25, 0.75, 1.25, 1.75, 0.25, 0.75, 1.25,
    1.75, 0.25, 0.75, 1.25, 1.75, 2.25, 2.75, 3.25, 3.75, 4.25, 4.75, 0.25, 0.75,
    1.25, 1.75, 2.25, 2.75, 3.25, 3.75, 4.25, 4.75, 0.25, 0.75, 1.25, 1.75, 2.25,
    2.75, 3.25, 3.75, 4.25, 4.75, 0.25, 0.75, 1.25, 1.75, 2.25, 2.75, 3.25, 3.75,
    4.25, 4.75, 0.25, 0.75, 1.25, 1.75, 0.25, 0.75, 1.25, 1.75, 0.25, 0.75, 1.25,
    1.75, 0.25, 0.75, 1.25, 1.75, 0.25, 0.75, 1.25, 1.75, 0.25, 0.75, 1.25, 1.75,
    0.25, 0.75, 1.25, 1.75, 2.25, 2.75, 3.25, 3.75, 4.25, 4.75, 0.25, 0.75, 1.25,
    1.75, 2.25, 2.75, 3.25, 3.75, 4.25, 4.75, 0.25, 0.75, 1.25, 1.75, 2.25, 2.75,
    3.25, 3.75, 4.25, 4.75, 0.25, 0.75, 1.25, 1.75, 2.25, 2.75, 3.25, 3.75, 4.25,
    4.75, 0.25, 0.75, 1.25, 1.75, 0.25, 0.75, 1.25, 1.75, 0.25, 0.75, 1.25, 1.75,
    0.25, 0.75, 1.25, 1.75, 0.25, 0.75, 1.25, 1.75, 0.25, 0.75, 1.25, 1.75 }
};
```

#### lib_properties.txt
```
For manual assignment to hardware configuration please
add the following additional include directories:

\Logical\MATLAB_includes\R2021b\

And the following additional build options:

-lm -D RT_MALLOC -D MODEL=cyklovac_BB -D NUMST=1 -D NCSTATES=0 -D HAVESTDIO -D RT -D USE_RTMODEL -D CLASSIC_INTERFACE=0 -D ALLOCATIONFCN=1 -D TID01EQ=0 -D MAT_FILE=0 -D ONESTEPFCN=1 -D TERMFCN=1 -D MULTI_INSTANCE_CODE=1 -D INTEGER_CODE=0 -D MT=0
```

### Library Logical/Libraries/regulatory
